# EPICS substitutions: apps/plcApp/Db/torus_interlocks.substitutions
#
# torus_interlock.substitutions
#
# Author: Wesley Moore (wmoore@jlab.org)
# Date:   July 2016
#

file "db/torus_bi_generic.db" {
    pattern{ PLCID, P, R, TAG, ZNAM, ONAM, ZSV, OSV, DESC }
    # Section 1, Hardwired Interlocks
    { PLC_TORUS, B_TORUS:, MPS:, LHe_Liquid_Level,    Ok, Fault, NO_ALARM, MAJOR, "LHe Liquid Level" }
    { PLC_TORUS, B_TORUS:, MPS:, VCL_Lead_T,          Ok, Fault, NO_ALARM, MAJOR, "Vapor Cooled Lead Temp" }
    { PLC_TORUS, B_TORUS:, MPS:, Watchdog,            Ok, Fault, NO_ALARM, MAJOR, "Chassis Watchdog" }
    { PLC_TORUS, B_TORUS:, MPS:, Lead_Water_Flow,     Ok, Fault, NO_ALARM, MAJOR, "Current Lead Water Flow" }
    { PLC_TORUS, B_TORUS:, MPS:, VT_Cable_Intlck      Ok, Fault, NO_ALARM, MAJOR, "VT Cable Intlk" }
    { PLC_TORUS, B_TORUS:, MPS:, System_Cable_Intlck, Ok, Fault, NO_ALARM, MAJOR, "System Cable Intlk" }
    { PLC_TORUS, B_TORUS:, MPS:, QD_Sum1,             Ok, Fault, NO_ALARM, MAJOR, "QD.Sum1 (ch1-4), dV>100mV" }
    { PLC_TORUS, B_TORUS:, MPS:, QD_Sum2,             Ok, Fault, NO_ALARM, MAJOR, "QD.Sum2 (ch5-8), dV>100mV,80mV" }
    { PLC_TORUS, B_TORUS:, MPS:, QD_Sum3,             Ok, Fault, NO_ALARM, MAJOR, "QD.Sum3 (ch9), dV>200mV" }
    { PLC_TORUS, B_TORUS:, MPS:, PLC_Fast_Dump,       Ok, Fault, NO_ALARM, MAJOR, "PLC Fast Dump Sum" }
    # Section 2, PLC Fast Dump Interlocks
    { PLC_TORUS, B_TORUS:, MPS:, EPICS_FastDump,      Ok, Fault, NO_ALARM, MAJOR, "EPICS Fast Dump Button" }
    { PLC_TORUS, B_TORUS:, MPS:, Hard_Overcurrent,    Ok, Fault, NO_ALARM, MAJOR, "Current Limit" }
    { PLC_TORUS, B_TORUS:, MPS:, RampDown_Fail,       Ok, Fault, NO_ALARM, MAJOR, "Ramp Down Fail" }
    { PLC_TORUS, B_TORUS:, MPS:, FIRE,                Ok, Fault, NO_ALARM, MAJOR, "VESDA Fire Detection" }
    { PLC_TORUS, B_TORUS:, MPS:, Soft_Quench_2nd,     Ok, Fault, NO_ALARM, MAJOR, "SW Quench, 2nd Threshold" }
    { PLC_TORUS, B_TORUS:, MPS:, UPS_Battery_Low,     Ok, Fault, NO_ALARM, MAJOR, "UPS Battery Low" }
    { PLC_TORUS, B_TORUS:, MPS:, ESR_INTLCK,          Ok, Fault, NO_ALARM, MAJOR, "ESR Fault" }
    # Section 3, PLC Controlled Ramp Down
    { PLC_TORUS, B_TORUS:, MPS:, Axial_Support_Interlock,     Ok, Fault, NO_ALARM, MAJOR, "Axial Support SG" }
    { PLC_TORUS, B_TORUS:, MPS:, DS_HB_SG_Interlock,  Ok, Fault, NO_ALARM, MAJOR, "DS Hex Beam SG" }
    { PLC_TORUS, B_TORUS:, MPS:, US_HB_SG_Interlock,  Ok, Fault, NO_ALARM, MAJOR, "US Hex Beam SG" }
    { PLC_TORUS, B_TORUS:, MPS:, CCM_LoadCell_Interlock,      Ok, Fault, NO_ALARM, MAJOR, "CCM Load Cell" }
    { PLC_TORUS, B_TORUS:, MPS:, VerticalSupport_Interlock,   Ok, Fault, NO_ALARM, MAJOR, "Vertical Support" }
    { PLC_TORUS, B_TORUS:, MPS:, Soft_Quench_1st,     Ok, Fault, NO_ALARM, MAJOR, "SW Quench" }
    { PLC_TORUS, B_TORUS:, MPS:, Vacuum_Interlock,    Ok, Fault, NO_ALARM, MAJOR, "Vacuum" }
    { PLC_TORUS, B_TORUS:, MPS:, EPICS_Watchdog_Fail, Ok, Fault, NO_ALARM, MAJOR, "EPICS Watchdog" }
    { PLC_TORUS, B_TORUS:, MPS:, Cryo_Interlock,      Ok, Fault, NO_ALARM, MAJOR, "Cryo(LHe LL/Pres,LN2 LL/Pres,VCL V/F/T)" }
    { PLC_TORUS, B_TORUS:, MPS:, Soft_Overcurrent,    Ok, Fault, NO_ALARM, MAJOR, "SW Current Limit (EPICS)" }
    { PLC_TORUS, B_TORUS:, MPS:, FastDAQ_Comm_Error,  Ok, Fault, NO_ALARM, MAJOR, "cRIO FastDAQ Comm" }
    { PLC_TORUS, B_TORUS:, MPS:, Splice_Overtemp,     Ok, Fault, NO_ALARM, MAJOR, "Splice(s) Over Temp" }
    # not an interlock, but used for alarm handler
    { PLC_TORUS, B_TORUS:, MPS:, cRIO_Comm_Error,     Ok, Fault, NO_ALARM, MAJOR, "cRIO LV Chassis Comm" }
    { PLC_TORUS, B_TORUS:, MPS:, FlagHeater_OutRange, Ok, Fault, NO_ALARM, MAJOR, "Temp Sensor Failed" }
}

file "db/torus_bi_renamed.db" {
    pattern{ PLCID, P, R, PV, TAG, ZNAM, ONAM, ZSV, OSV, DESC }
    { PLC_TORUS, B_TORUS:, MPS:, SOL_Quench,        Quench_Sol_Bool, Ok, Fault, NO_ALARM, MAJOR, "Solenoid Fast Dump, SW Quench Detection" }
    { PLC_TORUS, B_TORUS:, MPS:, VCL_A_Flow,        CryoSum[0], Ok, Fault, NO_ALARM, MAJOR, "VCL A FLow" }
    { PLC_TORUS, B_TORUS:, MPS:, VCL_B_Flow,        CryoSum[1], Ok, Fault, NO_ALARM, MAJOR, "VCL B FLow" }
    { PLC_TORUS, B_TORUS:, MPS:, VCL_A_Overtemp,    CryoSum[2], Ok, Fault, NO_ALARM, MAJOR, "VCL A Over Temp (TD8121A)" }
    { PLC_TORUS, B_TORUS:, MPS:, VCL_B_Overtemp,    CryoSum[3], Ok, Fault, NO_ALARM, MAJOR, "VCL B Over Temp (TD8121B)" }
    { PLC_TORUS, B_TORUS:, MPS:, WCL_A_Overtemp,    CryoSum[4], Ok, Fault, NO_ALARM, MAJOR, "WCL A Over Temp" }
    { PLC_TORUS, B_TORUS:, MPS:, WCL_B_Overtemp,    CryoSum[5], Ok, Fault, NO_ALARM, MAJOR, "WCL B Over Temp" }
    { PLC_TORUS, B_TORUS:, MPS:, LHe_Tank_Overpres, CryoSum[6], Ok, Fault, NO_ALARM, MAJOR, "LHe Tank Over Pres (PT8120)" }
    { PLC_TORUS, B_TORUS:, MPS:, SCC_Underpres,     CryoSum[7], Ok, Fault, NO_ALARM, MAJOR, "SuperCritical CCT Under Pres (PT8111)" }
    { PLC_TORUS, B_TORUS:, MPS:, LHe_LL_Low_DP,     CryoSum[8], Ok, Fault, NO_ALARM, MAJOR, "LHe Liquid Level Low (LL8120DP)" }
    { PLC_TORUS, B_TORUS:, MPS:, LHe_LL_Low_SC,     CryoSum[9], Ok, Fault, NO_ALARM, MAJOR, "LHe Liquid Level Low (LL8120SC)" }
}

file "db/torus_bo_generic.db" {
    pattern{ PLCID, P, R, TAG, ZNAM, ONAM, DESC }
    # Section 4, Comm Resets
    # TODO: multiples of CryoCon_Reset_PB
    { PLC_TORUS, B_TORUS:, MPS:, CryoCon_Reset_PB,    "", Reset, "Reset CryoCon Comm" }
    { PLC_TORUS, B_TORUS:, MPS:, LampTestReset,       "", Reset, "Reset CryoCon Comm" }
}

#
# SOE Timestamps (epoch)
#
file "db/datatype_soe.db" {
    pattern{ PLCID, P, R, PV, TAG, EGU }
    # LOWER
    { PLC_TORUS, B_TORUS:, MPS:, TSL_VCL_Lead_T,        Torus_EN2T2:7:I.Timestamp[0].OffOn[0],  "epoch" }
    { PLC_TORUS, B_TORUS:, MPS:, TSL_LHe_LL1,           Torus_EN2T2:7:I.Timestamp[1].OffOn[0],  "epoch" }
    # 2 - Spare
    # 3 - Spare
    # 4 - Spare
    # 5 - Spare
    { PLC_TORUS, B_TORUS:, MPS:, TSL_PLC_Fast_Dump,     Torus_EN2T2:7:I.Timestamp[6].OffOn[0],  "epoch" }
    # 7 - Spare
    { PLC_TORUS, B_TORUS:, MPS:, TSL_Watchdog,          Torus_EN2T2:7:I.Timestamp[8].OffOn[0],  "epoch" }
    { PLC_TORUS, B_TORUS:, MPS:, TSL_Lead_Water_Flow,   Torus_EN2T2:7:I.Timestamp[9].OffOn[0],  "epoch" }
    { PLC_TORUS, B_TORUS:, MPS:, TSL_VT_Cable,          Torus_EN2T2:7:I.Timestamp[10].OffOn[0], "epoch" }
    { PLC_TORUS, B_TORUS:, MPS:, TSL_System_Cable,      Torus_EN2T2:7:I.Timestamp[11].OffOn[0], "epoch" }
    { PLC_TORUS, B_TORUS:, MPS:, TSL_QD1_Sum,           Torus_EN2T2:7:I.Timestamp[12].OffOn[0], "epoch" }
    { PLC_TORUS, B_TORUS:, MPS:, TSL_QD2_Sum,           Torus_EN2T2:7:I.Timestamp[13].OffOn[0], "epoch" }
    { PLC_TORUS, B_TORUS:, MPS:, TSL_QD3_Sum,           Torus_EN2T2:7:I.Timestamp[14].OffOn[0], "epoch" }
    # 15 - Spare
    # UPPER
    { PLC_TORUS, B_TORUS:, MPS:, TSU_VCL_Lead_T,        Torus_EN2T2:7:I.Timestamp[0].OffOn[1],  "epoch" }
    { PLC_TORUS, B_TORUS:, MPS:, TSU_LHe_LL1,           Torus_EN2T2:7:I.Timestamp[1].OffOn[1],  "epoch" }
    # 2 - Spare
    # 3 - Spare
    # 4 - Spare
    # 5 - Spare
    { PLC_TORUS, B_TORUS:, MPS:, TSU_PLC_Fast_Dump,     Torus_EN2T2:7:I.Timestamp[6].OffOn[1],  "epoch" }
    # 7 - Spare
    { PLC_TORUS, B_TORUS:, MPS:, TSU_Watchdog,          Torus_EN2T2:7:I.Timestamp[8].OffOn[1],  "epoch" }
    { PLC_TORUS, B_TORUS:, MPS:, TSU_Lead_Water_Flow,   Torus_EN2T2:7:I.Timestamp[9].OffOn[1],  "epoch" }
    { PLC_TORUS, B_TORUS:, MPS:, TSU_VT_Cable,          Torus_EN2T2:7:I.Timestamp[10].OffOn[1], "epoch" }
    { PLC_TORUS, B_TORUS:, MPS:, TSU_System_Cable,      Torus_EN2T2:7:I.Timestamp[11].OffOn[1], "epoch" }
    { PLC_TORUS, B_TORUS:, MPS:, TSU_QD1_Sum,           Torus_EN2T2:7:I.Timestamp[12].OffOn[1], "epoch" }
    { PLC_TORUS, B_TORUS:, MPS:, TSU_QD2_Sum,           Torus_EN2T2:7:I.Timestamp[13].OffOn[1], "epoch" }
    { PLC_TORUS, B_TORUS:, MPS:, TSU_QD3_Sum,           Torus_EN2T2:7:I.Timestamp[14].OffOn[1], "epoch" }
    # 15 - Spare
}
